TYPE ST_EL2904 :
STRUCT
	//--------------------------------------------------------------------------------------------------------
	sTerminalName                                           :   STRING(200):= 'EL2904 | 4-Channel Digital Output';
	//=============================================================================================================
	// TERMINAL - EL2904	4-Channel Digital Output Terminal	 (Term 6)
	qEnableAirSupply_PSR1 					AT %Q*			: 	BOOL;	// EL2904 channel 1
	qResetAirSupply_PSR2					AT %Q* 			: 	BOOL;	// EL2904 channel 2
	qLockMainDoor             				AT %Q*	 		: 	BOOL;	// EL2904 channel 3 			
	qEL2904_Ch4      						AT %Q*	 		: 	BOOL;	// EL2904 channel 4 
	
	stTerminalInfo											: 	ST_Terminal_Info;
	
END_STRUCT
END_TYPE

(* stored: Version 1.1.0.1, ProductVersion 3.1.4024.13
   DUT ST_EL2904: Id {5f364899-56b6-4e28-b671-caca93aac3ae} *)
